(* IEC 61131-3 sources: RL_MAR/experiments/comparison/llm4plc/results/gpt-4o_20260507_114630/20260507_115703, 1 file *)

(* ---- generated_code_iteration_0.st ---- *)
plaintext
START_ST
FUNCTION_BLOCK WastewaterControl
VAR_INPUT
    InFlow : REAL; // Inlet flow rate
    OutFlow : REAL; // Outlet flow rate
    pH : REAL; // pH level
    TankLvl : REAL; // Tank level
END_VAR

VAR_OUTPUT
    Pump1 : BOOL; // Control for Pump1
    Pump2 : BOOL; // Control for Pump2
    Valve1 : BOOL; // Control for Valve1
    Valve2 : BOOL; // Control for Valve2
END_VAR

VAR
    state : INT := 0; // Current state of the FSM
    prevState : INT := -1; // Previous state of the FSM
    LowInFlow : REAL := 100.0; // Threshold for low inlet flow
    HighOutFlow : REAL := 90.0; // Threshold for high outlet flow
    DesiredPH : REAL := 7.0; // Threshold for pH adjustment
    HighTankLvl : REAL := 80.0; // Threshold for high tank level
END_VAR

// Main logic of the function block
IF state = 0 THEN
    // STATE 0: INITIALIZE
    Pump1 := FALSE;
    Pump2 := FALSE;
    Valve1 := FALSE;
    Valve2 := FALSE;
    prevState := state;
    state := 1; // Transition to STATE 1

ELSIF state = 1 THEN
    // STATE 1: MONITOR AND CONTROL PUMP1
    IF InFlow < LowInFlow THEN
        Pump1 := TRUE;
    ELSE
        Pump1 := FALSE;
    END_IF;
    prevState := state;
    state := 2; // Transition to STATE 2

ELSIF state = 2 THEN
    // STATE 2: MONITOR AND CONTROL PUMP2
    IF OutFlow > HighOutFlow THEN
        Pump2 := TRUE;
    ELSE
        Pump2 := FALSE;
    END_IF;
    prevState := state;
    state := 3; // Transition to STATE 3

ELSIF state = 3 THEN
    // STATE 3: MONITOR AND CONTROL VALVE1
    IF pH < DesiredPH THEN
        Valve1 := TRUE;
    ELSE
        Valve1 := FALSE;
    END_IF;
    prevState := state;
    state := 4; // Transition to STATE 4

ELSIF state = 4 THEN
    // STATE 4: MONITOR AND CONTROL VALVE2
    IF TankLvl > HighTankLvl THEN
        Valve2 := TRUE;
    ELSE
        Valve2 := FALSE;
    END_IF;
    prevState := state;
    state := 1; // Transition back to STATE 1

END_IF;
END_FUNCTION_BLOCK
END_ST
